////////////////////////////////////////////////////////////////////////////////////////////////////////////
(*	TKMatik
	Blok funkcyjny, sterujacy falownikiem firmy Lenze model:i550
	v.1.3 16.01.2019
	v.1.4 22.08.2019
	v.1.5 29.07.2020
	Wymagane pliki: E_Station (ENUM)
	Data modyfikacji: 29.07.2020
	
	--->Obsluga bloku:
	Blok umozliwia sterownie falownikiem Lenze i550 w trybie manulanym i automatycznym
	*TRYB AUTOMATYCZNY*
	Po podaniu sygnalu wysokiego na wejscie bEnable rozoczyna sie procedura uruchamiania falownika
	Wejscie bRun umozliwiaja odpowiednio uruchomienie silnika i jego zatrzymanie 
	Wejscie bReset umozliwa wykonanie procedury resetu bloku i bledu falownika
	Wejscia iMinSpeed_rpm oraz iMaxSpeed_rpm pozwalaja na programowe ograniczenie obrotow silnika
	Wejscie iSpeed sluzy zadawania wartosci predkosci
	Mozliwa jest rowniez zmiana kierunku obrotow silnika przy pomocy wejscia bDirection
	*TRYB MANULANY*
	Sterowanie w trybie manulanym opiera sie o wykrywanie czasu przyciniecia przyciku
	Dla krotkiego przycisniecia wykonywany jest ruch silnika o krok ktorego czas musi byc zadany na wejscie bloku - opcje ta mozna dezaktywowac wejsciem bStepModeNotActive
	Dla dlugiego przycisniecia ruch jest wykonywany do czasu zaprzestania naciskania przycisku
	
	
	Wejscia bloku, ktore nalezy polinkowac ze zmiennymi falownika:
		-uiErrorCode
		-uiStatusWord
		-ActualSpeed 
	Wyjscia bloku, ktore nalezy polinkowac ze zmiennymi falownika:
		-uiControlWord
		-iSendVelocity
*)
////////////////////////////////////////////////////////////////////////////////////////////////////////////

FUNCTION_BLOCK FB_LenzeInverter

VAR_INPUT
	bEStop														: BOOL;													// Pozwolenie na prace bloku z SAFETY (TRUE-maszyna gotowa do pracy FALSE-brak pozolenia na prace)
	bWcState													: BOOL;													// Zmienna WcState - TRUE w przypadku odebrania niewlasciwej ramki EtherCAT
	bDirection													: BOOL;													// Kierunek obrotow silnika 
	iMinSpeed_rpm												: INT				:= 1000;							// Minimalna prędkość obrotowa
	iMaxSpeed_rpm												: INT				:= 2840;							// Maksymalna prędkość obrotowa
	iRatedSynchornousRPM										: INT				:= 3000;							// Predkosc synchorniczna (wzor: RatedSynchronousRPM = 60 * Frequency / NumberOfPolePair)
	iRatedRotorRPM												: INT				:= 2840;							// Znamionowe obroty silnika
	rGear														: REAL;													// Przekładnia
	iIndex														: INT;													// Indeks falownika
	bEnable														: BOOL;													// Uruchomienie bloku
	bRun														: BOOL;													// Komenda na uruchomienie 
	bReset														: BOOL;													// Reset falownika po bledzie
	bManualMode													: BOOL;													// Tryb manualny
	bJogForward													: BOOL;													// Komenda na ruch w kierunku dodatnim 
	bJogBackward												: BOOL;													// Komenda na ruch w kierunku ujemnym 
	bDeactivateStepMode											: BOOL;													// Zmienna dezaktywujaca przesuwanie silnika o krok po nacisnieciu JOGa
	uiErrorCode 				(*Devices*)						: UINT;													// Kod bledu falownika
	bFullConveyorStopSensor										: BOOL;													// Zatrzymanie transportera ze względu zapełnienia
	uiStatusWord				(*Devices*)						: UINT;													// Status wysylany z falownika
	iActualSpeedIn				(*Devices*)						: INT;													// Zmienna z falownika przepisana na wyjscie do zmiennej QiActualSpeed
	tTimeOfJog													: TIME				:= T#2S;
	iStationIndex												: UDINT;												// Numer stacji 
	sStationName												: WSTRING;												// Nazwa stacji
	iSpeed														: INT;													// Predkosc zadana przypisana do zmiennej Qn_SV wysylanej do falownika  
END_VAR                                                                         			                    		
VAR_OUTPUT                                                                      			                    		
	eState														: E_Station;											// Stan pracy bloku
	
	bError														: BOOL;													// Blad falownika
	udiErrorID													: UDINT;												// Nr błędu bloku funkcyjnego
	sErrorDescription											: STRING(200);											// Opis błędu
	sErrorDescription2											: STRING(200);											// Opis błędu
	sErrorStationName											: STRING;												// Nazwa stacji
	udiStationID												: UDINT;				// Nr stacji	
	uiControlWord(*Wymaga przypisania do urządzenia*)			: UINT;													// ControlWord wysylany do falownika 
	iSendVelocity(*Wymaga przypisania do urządzenia*)			: INT;													// Wartosc predkosci zadanej wysylanej do falownika
	iActualSpeedOut												: INT;													// Wartosc predkosci akutalnej przepisanej z wyjscia
	iSlipCorrector												: INT;													// Wspolczynnik korygujacy wartosc poslizgu
	iManualStep													: INT;
END_VAR                                     					
VAR                                         					
	rtRun														: R_TRIG;												// Triger rozpoczynajacy obrot osi silnika
	ftReset														: F_TRIG;												// Triger zbocza opadajacego resetu
	rtInvertDirection											: R_TRIG;												// Triger zmieniajacy kierunek obrotu osi silnika
	ftInvertDirection											: F_TRIG; 												// Triger zbocza opadajacego od zmiany kierunku                                      		                                                                                                          		                 											                                		
	rtJogForward												: R_TRIG;												// Trigger wykrywajacy zbocze narasatace komendy ruchu w kierunku dodatnim w trybie manulanym
	rtJogBackward												: R_TRIG;												// Trigger wykrywajacy zbocze narasatace komendy ruchu w kierunku ujemnym w trybie manulanym
	ftJogForward												: F_TRIG;												// Trigger wykrywajacy zbocze opadajace komendy ruchu w kierunku dodatnim w trybie manulanym
	ftJogBackward												: F_TRIG;												// Trigger wykrywajacy zbocze opadajace komendy ruchu w kierunku ujemnym w trybie manulanym
                                     					
	tonTimeOfJog												: TON;													// Timer odliczajacy czas trwania ruchu silnika w trybie manualnym
	tonPressing													: TON;													// Timer odliczajacy czas nacisniecia przycisku w trybie manulanym
	
    iCalculateVelocity											: INT;													// Wartosc predkosci wykorzystwanej do obliczen w bloku                                  	                                                                		
	
	bCheckInitTimeError											: BOOL;													// Blad oczekiwania na odpowiedz falownika
	tonCheckInitTime											: TON;													// Timer odliczajacy czas odpowiedzi falownika
	
	bWcStateError												: BOOL;													// Blad zmiennej WcState - odczytanie blednej ramki danych przez urzadzenie EtherCAT
	
	bLenzeReadiness												: BOOL;													// Gotowosc falownika do pracy na podstawie bitu StatusWord --> SwitchedOn
	bLenzeReadinessError										: BOOL;													// Blad zwiazany z utraceniem gotowosci do pracy przez falownik
	bFullConveyorError											: BOOL;														// Blad zwiazany z przepełnieniem transportera
	
	
	iPreparingStep												: INT;													// Krok procedury przygotowania do pracy falownika
	
	
	(*Zmienne ControlWord*)
	bSwitchOn													: BOOL;													// Zalacz falownik do trybu gotowsci
	bEnableVoltage												: BOOL;													// Zalacz zasilanie na zaciski falownika
	bQuickStop													: BOOL;													// Bezpieczne zatrzymanie
	bEnableOperation											: BOOL;													// Rozpoczecie pracy falownika
	bOperationModeSpecific1										: BOOL;
	bOperationModeSpecific2										: BOOL;
	bOperationModeSpecific3										: BOOL;
	bFaultReset													: BOOL;													// Reset bledu
	bHalt														: BOOL;													// Zatrzymanie procesowe
	bOperationModeSpecific4										: BOOL;
	bReserved1													: BOOL;
	bReserved2													: BOOL;
	bReserved3													: BOOL;
	bReserved4													: BOOL;
	bHoldingBrakeRelease										: BOOL;
	bReserved5													: BOOL;
	                                        					
	(*Zmienne StatusWord*)                  					
	bReadyToSwitchOn											: BOOL;													// Gotowy na zalaczenie do trybu gotowosci
	bSwitchedOn													: BOOL;													// Zalaczony w tryb gotowosci do pracy
	bOperationEnabled											: BOOL;													// Wykonywanie pracy
	bFaultActive												: BOOL;													// Akytwny blad falownika
	bVoltageEnabled												: BOOL;													// Zalaczone zasilanie na zaciski falownika
	bQuickStopActive											: BOOL;													// Aktywne bezpieczne zatrzymanie				
	bSwitchOnDisabled											: BOOL;													// Tryb nieaktywnosci falownika	
	bWarningActive												: BOOL;													// Aktywne ostrzezenie falownika
	bDeactiveRPDOs												: BOOL;
	bRemote														: BOOL;													// Mozliwosc wykonyania operacji
	bTargetReached												: BOOL;													// Osiagniecie predkosci zadanej
	bInternalLimitActive										: BOOL;
	bReserved6													: BOOL;
	bReserved7													: BOOL;
	bBreakeReleased												: BOOL;
	bSTONotActive												: BOOL;													// Bezpieczne zatrzymanie nieaktywne
	
	rLenzeGear													: REAL;
	
			//Zmienne od EVENTLOGGER
	bAlarmInit 						: BOOL := TRUE; 
	nAlarmNumerator					: INT;
	arfbAlarm						: ARRAY[0..19] OF  FB_TcAlarm;		//Tablica bloczków błędów
	fbSourceInfo 					: FB_TcSourceInfo;
	iSourceInfo						: I_TcSourceInfo;
	sAlarmTest						: STRING;
	//Koniec zmiennych od EVENTLOGGER
END_VAR

VAR_IN_OUT
 
END_VAR


(*Status WORD:													
	Bit 0: Ready to switch on
	Bit 1: Switched on
	Bit 2: Operation enabled
	Bit 3: Fault active
	Bit 4: Voltage enabled
	Bit 5: Quick stop
	Bit 6: Switch on disabled
	Bit 7: Warning active
	Bit 8: Deactivate RPDOs
	Bit 9: Remote
	Bit 10: Target speed reached
	Bit 11: Internal limit active
	Bit 12: Reserved
	Bit 13: Reserved
	Bit 14: Brake released
	Bit 15: Safe torque off (STO) not active*)
				
	(*Control WORD:
	Bit 0: Switch On
	Bit 1: Enable Voltage
	Bit 2: Activate quick Stop
	Bit 3: Enable operation
	Bit 4: Operation mode specific
	Bit 5: Operation mode specific
	Bit 6: Operation mode specific
	Bit 7: Fault reset
	Bit 8: Halt
	Bit 9: Operation mode specific
	Bit 10: Reserved
	Bit 11: Reserved
	Bit 12: Reserved
	Bit 13: Reserved
	Bit 14: Holding brake release
	Bit 15: Reserved*)

ACT_EStop();
ACT_StatusWord();																										// Przypisanie bitow StatusWorda do zmiennych
ACT_ErrorHandling();
aStationID();

rtRun															(CLK:= bRun);
rtJogForward													(CLK:= bJogForward);
rtJogBackward													(CLK:= bJogBackward);
ftJogForward													(CLK:= bJogForward);
ftJogBackward													(CLK:= bJogBackward);
                                                               
                                                                
IF 	NOT bEnable 												AND 
	bEStop 														AND  
	eState <> E_Station.eAborting 								AND 
	eState <> E_Station.eAborting 								THEN
	
	eState:= E_Station.ePreparingToDisable;
END_IF


		
CASE eState OF
	
	E_Station.ePreparingToDisable: (*Przygotowanie do wylaczenia*)
	
		bQuickStop 												:= FALSE;
		bEnableVoltage											:= FALSE;
		bSwitchOn												:= FALSE;
		bEnableOperation 										:= FALSE;
		bFaultReset												:= FALSE;
		tonTimeOfJog.IN											:= FALSE;
		tonPressing.IN											:= FALSE;
		iPreparingStep											:= 0;
		iManualStep												:= 0;
		
		bLenzeReadinessError									:= FALSE;
		bFullConveyorError										:= FALSE;
		bWcStateError											:= FALSE;
		bCheckInitTimeError										:= FALSE;
		                                         
		eState:= E_Station.eDisabled;

		
	E_Station.eDisabled: (*Stan nieaktywnosci falowika*)
	
		IF bEnable THEN																									// Rozpoczecie proceduru uruchomienia falownika 								
			eState:= E_Station.ePreparingToReady;	                                		                                							
		END_IF                                      		                                							
	
			                                    		                                													
	E_Station.ePreparingToReady: (*Przygotwanie do gotowosci*)
	
	
		CASE iPreparingStep OF
			0:
				bSwitchOn										:= FALSE;
			    bEnableVoltage	                                := FALSE;
			    bQuickStop		                                := FALSE;
			    bEnableOperation                                := FALSE;
				iPreparingStep:= 10;
				
				IF bSwitchedOn THEN
					iPreparingStep:= 30;
				END_IF
				
			10:
				IF bSwitchOnDisabled THEN
					bEnableVoltage								:= TRUE;
					bQuickStop									:= TRUE;
					iPreparingStep:= 20;
				END_IF
			
			20:
				IF bReadyToSwitchOn THEN
					bSwitchOn									:= TRUE;
					iPreparingStep:= 30;
				END_IF
			
			30:
				IF bSwitchedOn THEN
					iPreparingStep:= 0;
					eState:= E_Station.eReady;
				END_IF
				
				
		END_CASE
	
			
	E_Station.eReady:	(*Gotowosc i oczekiwanie na komendy*)

		IF rtRun.Q THEN
			bEnableOperation									:= TRUE;
			eState:= E_Station.eStarting;
		END_IF
		
		IF bManualMode THEN
			iManualStep:= 0;
			eState:= E_Station.eManualMovement;
		END_IF
														
		
		
	E_Station.eStarting: (*Stan rozpoczynania pracy falownika*)
	
		IF bOperationEnabled THEN
			eState:= E_Station.eRunning;
		END_IF
		
		IF NOT bRun THEN
			bEnableOperation									:= FALSE;									
			eState:= E_Station.eStopping;
		END_IF
		
				
	E_Station.eRunning: (*Stan wykonywania pracy falownika*)
	
		IF NOT bRun THEN
			bEnableOperation									:= FALSE;									
			eState:= E_Station.eStopping;
		END_IF
		
			
	E_Station.eStopping:
	
		IF NOT bOperationEnabled THEN
			eState:= E_Station.eReady;
		END_IF
		
				
	E_Station.eAborting: (*Stan bezpiecznego zatrzymywania silnika*)	
	
		bQuickStop 												:= FALSE;
	    bEnableVoltage											:= FALSE;
	    bSwitchOn												:= FALSE;
		bEnableOperation 										:= FALSE;
		
		tonTimeOfJog.IN											:= FALSE;
		tonPressing.IN											:= FALSE;
		iManualStep												:= 0;
		iPreparingStep											:= 0;
		
		
		eState:= E_Station.eAborted;
		
		
	E_Station.eAborted: (*Stan bezpiecznego zatrzymania silnika*)
	                              			
		IF bEstop THEN
			IF NOT bError THEN
				IF bEnable THEN
					eState:= E_Station.ePreparingToReady;
				ELSE
					eState:= E_Station.ePreparingToDisable;
				END_IF
			ELSE 
				eState:= E_Station.eError;	
			END_IF	
		END_IF
		
					
	E_Station.eError: (*Stan bledu*)
													
		bQuickStop 												:= FALSE;
		bEnableVoltage											:= FALSE;
		bSwitchOn												:= FALSE;
		bEnableOperation 										:= FALSE;
		
		tonTimeOfJog.IN											:= FALSE;
		tonPressing.IN											:= FALSE;
		iManualStep												:= 0;
		iPreparingStep											:= 0;

		IF bReset THEN
			IF bCheckInitTimeError THEN
				bCheckInitTimeError								:= FALSE;
			END_IF
			IF bWcStateError THEN
				bWcStateError									:= FALSE;
			END_IF
			IF bLenzeReadinessError THEN
				bLenzeReadinessError							:= FALSE;
			END_IF
			IF 	bFullConveyorError	THEN
				bFullConveyorError								:= FALSE;
			END_IF
		END_IF
		
		bFaultReset												:= bReset; 

		
		IF NOT bError THEN 
			
			bFaultReset											:= FALSE;
		
			eState:= E_Station.ePreparingToReady;	
				
		END_IF
		
		
	E_Station.eManualMovement: (*Stan wykonywania ruchow manualnych*)
		
		ACT_ManualMovements();
		
									
END_CASE



IF ABS(iActualSpeedIn) > iSlipCorrector THEN
	IF iActualSpeedIn > 0 THEN
		iActualSpeedOut													:= (iActualSpeedIn - iSlipCorrector) / REAL_TO_INT(rGear);					// Przepisanie wartosci z wejscia bloku na jego wyjscie		
	ELSE
		iActualSpeedOut													:= (iActualSpeedIn + iSlipCorrector) / REAL_TO_INT(rGear);					// Przepisanie wartosci z wejscia bloku na jego wyjscie	
	END_IF
ELSE
	iActualSpeedOut													:= 0;
END_IF										


ACT_Calculations();	
ACT_ControlWord();																									//Przypisanie zmiennych do bitow ControlWorda


tonPressing();																								
tonTimeOfJog();

ACTION ACT_Calculations:
                                                    		
(*IF ABS(iSpeed) < iMinSpeed_rpm THEN																						// Warunki programowaego ograniczenia predkosci do wartosci min i max
	iSpeed 														:= iMinSpeed_rpm;
END_IF                                                  		
IF ABS(iSpeed) > iMaxSpeed_rpm THEN                     		
	iSpeed														:= iMaxSpeed_rpm;
END_IF                                                  	
*)//dp
                                                   	
IF bDirection THEN																										                                    	
	iCalculateVelocity											:= -iSpeed;
ELSE                                                    	
	iCalculateVelocity											:= iSpeed;
END_IF

(*Ruchy manualne JOG definuja kierunek ruchu niezaleznie od bDirection*)		
IF bJogForward THEN
	iCalculateVelocity											:= iSpeed;
ELSIF bJogBackward THEN
	iCalculateVelocity											:= -iSpeed;
END_IF
	

iSlipCorrector													:= iRatedSynchornousRPM - iRatedRotorRPM;				// Obliczenie wspolczynnika korygujacego wartosc poslizgu


(*Kontrola poprawności parametryzacji przekładni*)
IF rGear < 1 THEN
	rLenzeGear													:= 1;
ELSE
	rLenzeGear													:= rGear;
END_IF


(*Korekcja wartosci zadanej predkosci o wartosc poslizgu*)
IF iCalculateVelocity >= 0 THEN
	iSendVelocity												:= (iCalculateVelocity * REAL_TO_INT(rLenzeGear)) + iSlipCorrector ;
ELSIF iCalculateVelocity <0 THEN
	iSendVelocity												:= (iCalculateVelocity * REAL_TO_INT(rLenzeGear)) - iSlipCorrector;
END_IF
END_ACTION

ACTION ACT_ControlWord:
uiControlWord.0 								:= bSwitchOn;
uiControlWord.1 								:= bEnableVoltage;
uiControlWord.2 								:= bQuickStop;
uiControlWord.3 								:= bEnableOperation;
uiControlWord.4 								:= bOperationModeSpecific1;
uiControlWord.5 								:= bOperationModeSpecific2;
uiControlWord.6 								:= bOperationModeSpecific3;
uiControlWord.7 								:= bFaultReset;
uiControlWord.8 								:= bHalt;
uiControlWord.9 								:= bOperationModeSpecific4;
uiControlWord.10 								:= bReserved1;
uiControlWord.11 								:= bReserved2;
uiControlWord.12 								:= bReserved3;
uiControlWord.13 								:= bReserved4;
uiControlWord.14 								:= bHoldingBrakeRelease;
uiControlWord.15 								:= bReserved5;
END_ACTION

ACTION ACT_ErrorHandling:
// Alarm_0580	580	Error	Zresetuj błąd na panelu falownika {0}
// Alarm_0581	581	Error	Błąd komunikacji z urządzeniem (WcState)
// Alarm_0582	582	Error	Utracono gotowość falownika do pracy
// Alarm_0583	583	Error	Przekroczenie czasu oczekiwania na odpowiedź falownika
// Alarm_0584	584	Error	Przepełnienie

IF bAlarmInit THEN
    bAlarmInit := FALSE; 
	fbSourceInfo.Clear();
	fbSourceInfo.sName:=wsLiteral_TO_UTF8(sStationName);//'Machine';
	fbSourceInfo.nId:=iStationIndex;//2700;
	// Alarm_0580	580	Error	Zresetuj błąd na panelu falownika {0}
    arfbAlarm[0].CreateEx(stEventEntry := TC_EVENTS.AlarmClass.Alarm_0580, bWithConfirmation:= FALSE,  ipSourceInfo:= fbSourceInfo); 
	// Alarm_0581	581	Error	Błąd komunikacji z urządzeniem (WcState)
	arfbAlarm[1].CreateEx(stEventEntry := TC_EVENTS.AlarmClass.Alarm_0581, bWithConfirmation:= FALSE,  ipSourceInfo:= fbSourceInfo);
	// Alarm_0582	582	Error	Utracono gotowość falownika do pracy
	arfbAlarm[2].CreateEx(stEventEntry := TC_EVENTS.AlarmClass.Alarm_0582, bWithConfirmation:= FALSE,  ipSourceInfo:= fbSourceInfo);
	// Alarm_0583	583	Error	Przekroczenie czasu oczekiwania na odpowiedź falownika
	arfbAlarm[3].CreateEx(stEventEntry := TC_EVENTS.AlarmClass.Alarm_0583, bWithConfirmation:= FALSE,  ipSourceInfo:= fbSourceInfo);
	// Alarm_0584	584	Error	Przepełnienie
	arfbAlarm[4].CreateEx(stEventEntry := TC_EVENTS.AlarmClass.Alarm_0584, bWithConfirmation:= FALSE,  ipSourceInfo:= fbSourceInfo);
	
END_IF



tonCheckInitTime.IN												:= eState = E_Station.ePreparingToReady OR eState = E_Station.eStarting OR eState = E_Station.eStopping;																														
tonCheckInitTime.PT												:= T#5S;
tonCheckInitTime();                                     		

IF tonCheckInitTime.Q THEN
	bCheckInitTimeError											:= TRUE;
END_IF  

IF bWcState THEN
	bWcStateError												:= TRUE;
END_IF   

IF bFullConveyorStopSensor THEN
	bFullConveyorError:= TRUE;
END_IF

bLenzeReadiness													:= bSwitchedOn;

IF NOT bLenzeReadiness THEN
	IF 	eState = E_Station.eReady				OR
		eState = E_Station.eStarting			OR
		eState = E_Station.eRunning				OR
		eState = E_Station.eStopping			OR
		eState = E_Station.eManualMovement		THEN

		bLenzeReadinessError									:= TRUE;
		
	END_IF                                                		
END_IF    

                                         	                                                        	                                                     	
//bError															:= bFaultActive OR bCheckInitTimeError OR bWcStateError OR bLenzeReadinessError OR bFullConveyorError;

// Alarm_0580	580	Error	Zresetuj błąd na panelu falownika {0}
IF bFaultActive AND bEnable THEN
	arfbAlarm[0].ipArguments.Clear() .AddUInt(uiErrorCode);
		IF NOT arfbAlarm[0].bActive THEN		
			arfbAlarm[0].Raise(nTimeStamp:=0);
		END_IF
	ELSE	
		IF  arfbAlarm[0].bActive AND bReset THEN
			arfbAlarm[0].Clear(nTimeStamp:=0, bResetConfirmation:= FALSE);
		END_IF
// 	udiErrorID													:= 357;//uiErrorCode;
// 	sErrorDescription											:= 'Zresetuj błąd na panelu falownika.';
// 	sErrorDescription2											:= UINT_TO_STRING(uiErrorCode);
END_IF	
 // Alarm_0581	581	Error	Błąd komunikacji z urządzeniem (WcState)                                               	
IF bWcStateError AND bEnable THEN
	IF NOT arfbAlarm[1].bActive THEN		
			arfbAlarm[1].Raise(nTimeStamp:=0);
		END_IF
	ELSE	
		IF  arfbAlarm[1].bActive AND bReset THEN
			arfbAlarm[1].Clear(nTimeStamp:=0, bResetConfirmation:= FALSE);
		END_IF
// 	udiErrorID													:= 358;//INT_TO_UDINT(iIndex + 1) ;	
// 	sErrorDescription											:= 'Błąd komunikacji z urządzeniem (WcState)';
END_IF
// Alarm_0582	582	Error	Utracono gotowość falownika do pracy
IF bLenzeReadinessError AND bEnable THEN
		IF NOT arfbAlarm[2].bActive THEN		
			arfbAlarm[2].Raise(nTimeStamp:=0);
		END_IF
	ELSE	
		IF  arfbAlarm[2].bActive AND bReset THEN
			arfbAlarm[2].Clear(nTimeStamp:=0, bResetConfirmation:= FALSE);
		END_IF
// 	udiErrorID													:= 359;//INT_TO_UDINT(iIndex + 2) ;	
// 	sErrorDescription											:= 'Utracono gotowość falownika do pracy';
END_IF	
// Alarm_0583	583	Error	Przekroczenie czasu oczekiwania na odpowiedź falownika
IF bCheckInitTimeError AND bEnable THEN
		IF NOT arfbAlarm[3].bActive THEN		
			arfbAlarm[3].Raise(nTimeStamp:=0);
		END_IF
	ELSE	
		IF  arfbAlarm[3].bActive AND bReset THEN
			arfbAlarm[3].Clear(nTimeStamp:=0, bResetConfirmation:= FALSE);
		END_IF                             	
// 	udiErrorID													:= 360;//INT_TO_UDINT(iIndex  + 3) ;	
// 	sErrorDescription											:= 'Przekroczenie czasu oczekiwania na odpowiedź falownika';
END_IF	
// Alarm_0584	584	Error	Przepełnienie
IF bFullConveyorError AND bEnable  THEN
	IF NOT arfbAlarm[4].bActive THEN		
			arfbAlarm[4].Raise(nTimeStamp:=0);
		END_IF
	ELSE	
		IF  arfbAlarm[4].bActive AND bReset THEN
			arfbAlarm[4].Clear(nTimeStamp:=0, bResetConfirmation:= FALSE);
		END_IF
// 	udiErrorID													:= 361;//INT_TO_UDINT(iIndex  + 4) ;	
// 	sErrorDescription											:= 'Przepełnienie';
END_IF


	
IF NOT bEnable THEN
	bError														:= FALSE;
	udiErrorID													:= 0;
	sErrorDescription											:= ''; 
END_IF	

(*Wyświetlanie błedu na wyjściu*)
bError							:= FALSE;
FOR nAlarmNumerator := 0 TO 19 DO
	bError						:= bError OR arfbAlarm[nAlarmNumerator].bActive;
END_FOR
	
IF bError THEN

	IF 	eState = E_Station.ePreparingToReady    OR
	    eState = E_Station.eReady               OR      
	    eState = E_Station.eStarting			OR           
	    eState = E_Station.eRunning			    OR  
		eState = E_Station.eStopping			OR    
	   	eState = E_Station.eManualMovement      THEN
		
		eState													:= E_Station.eError;	
	END_IF
                                      
END_IF

IF NOT bError THEN
	udiErrorID													:= 0;
	//sErrorDescription											:= ""; 
	sErrorDescription											:= ''; 
END_IF





sErrorStationName:=WSTRING_TO_STRING(sStationName);
END_ACTION

ACTION ACT_EStop:
IF NOT bEStop THEN
	IF eState <> E_Station.eAborted THEN
		IF eState <> E_Station.eAborting THEN
			eState:= E_Station.eAborting;	
		END_IF
	END_IF
END_IF
END_ACTION

ACTION ACT_ManualMovements:
CASE iManualStep OF
			
	0: (*Oczekiwanie na zbocze narastajace komendy ruchu JOG*)
	
		bEnableOperation										:= bRun;
		
		IF rtJogForward.Q THEN
			tonPressing.IN										:= TRUE;
			tonPressing.PT										:= T#1S;
			iManualStep:= 10;
		END_IF
					
		IF rtJogBackward.Q THEN
			tonPressing.IN										:= TRUE;
			tonPressing.PT										:= T#1S;
			iManualStep:= 20;
		END_IF
		
	
	10: (*Oczekiwanie na zbocze opadajace komendy ruchu JOG w kierunku pozytywnym*)
	
		bEnableOperation												:= TRUE;
	                                                                	
		IF NOT bJogForward THEN	                                    	
			IF tonPressing.Q OR bDeactivateStepMode	THEN            	
				iManualStep:= 100;	
			ELSIF NOT tonPressing.Q AND NOT bDeactivateStepMode THEN	
				tonTimeOfJog.IN											:= TRUE;
				tonTimeOfJog.PT											:= tTimeOfJog;
				iManualStep:= 50;
			END_IF                                                  	
			tonPressing.IN												:= FALSE;
		END_IF
		
	
	20: (*Oczekiwanie na zbocze opadajace komendy ruchu JOG w kierunku negatywnym*)
		
		bEnableOperation												:= TRUE;
	                                                                	
		IF NOT bJogBackward THEN	                                    	
			IF tonPressing.Q OR bDeactivateStepMode	THEN            	
				iManualStep:= 100;	
			ELSIF NOT tonPressing.Q AND NOT bDeactivateStepMode THEN	
				tonTimeOfJog.IN											:= TRUE;
				tonTimeOfJog.PT											:= tTimeOfJog;
				iManualStep:= 50;
			END_IF                                                  	
			tonPressing.IN												:= FALSE;
		END_IF
		
	50: (*Oczekiwanie na odliczenie czasu kroku*)
	
		IF tonTimeOfJog.Q THEN
			tonTimeOfJog.IN												:= FALSE;
			iManualStep:= 100;
		END_IF
		
	100: (*Zakonczenie ruchu*)
	
		bEnableOperation												:= FALSE;
		iManualStep:= 0;	

END_CASE


IF NOT bManualMode THEN
	tonTimeOfJog.IN														:= FALSE;
	tonPressing.IN														:= FALSE;
	bEnableOperation													:= FALSE;
	iManualStep															:= 0;
	eState:= E_Station.eReady;
END_IF
END_ACTION

ACTION ACT_StatusWord:
bReadyToSwitchOn 								:= uiStatusWord.0;
bSwitchedOn 									:= uiStatusWord.1;
bOperationEnabled 								:= uiStatusWord.2;
bFaultActive 									:= uiStatusWord.3;
bVoltageEnabled 								:= uiStatusWord.4; 
bQuickStopActive 								:= uiStatusWord.5; 
bSwitchOnDisabled 								:= uiStatusWord.6;
bWarningActive 									:= uiStatusWord.7; 
bDeactiveRPDOs 									:= uiStatusWord.8; 
bRemote											:= uiStatusWord.9; 
bTargetReached									:= uiStatusWord.10;
bInternalLimitActive							:= uiStatusWord.11;
bReserved6										:= uiStatusWord.12;
bReserved7										:= uiStatusWord.13;
bBreakeReleased									:= uiStatusWord.14;
bSTONotActive									:= uiStatusWord.15;
END_ACTION

ACTION aStationID:
udiStationID	:=	iStationIndex;
END_ACTION

END_FUNCTION_BLOCK

(* stored: Version 1.1.0.1, ProductVersion 3.1.4026.13, FileIdentifier 9ad2ff281ca15bdc4701e5a91a6fd127a2ff6bba, FileSignature 7266ffc515f8d221687c75fdba088e1f67518c5d238bbab9f17c99c9903b828c719495a2eae69af3465cf855b77689457414dd553be6ef4fb2c18110e40bf5b4f4c678a4f04c66342ad6b635ebf4b1c8b74fe8689a8c66a332ec2c82a04ae904786038ab1bab508a29c2edceec5ad5bc1dc3aa1eea3bdab653c41812187d267dde7562c469d8f6f27775aa94d02276b55294e497f498f22daee374bcfc3cb06d760aadc96bcc2b21c3f5c0f0ac8dbe488ed612767664df79a9cee58243d12ab428a3689f0aa0222e8db84ccf62597463c89ddb4223b6820c1feb0da994420665123bedf30d52a9ae24a51afed12cf98888f7ec44261e6800110c49d66fb3e59e
   POU FB_LenzeInverter: Id {7d78c98b-d7e0-49c7-b6bc-7b71ac652246}, SpecialFunc None
   Action ACT_Calculations: Id {f6efc5c3-cb90-41f3-9e07-8c06c8560a5d}
   Action ACT_ControlWord: Id {b0bb2c43-b153-4ff8-8fd7-446ba91f7eec}
   Action ACT_ErrorHandling: Id {6326a32b-28ec-40d5-b8a8-82a14992ccb9}
   Action ACT_EStop: Id {f52ef56e-481b-4442-b7c7-52c588154dd9}
   Action ACT_ManualMovements: Id {58896d9f-cc56-4bdc-8390-4d53b4407917}
   Action ACT_StatusWord: Id {7cd6f049-ad3d-4440-ac74-13d1cd4616cc}
   Action aStationID: Id {6515a2a1-e0ce-4bb6-8f7c-0794d2270d0d} *)
